Staubli VAL3: loadTemplate.pgx

program loadTemplate()
begin
  // load the default instruction
  events:libLoad("Disk://..//templates/instruction")
  delay(0)
end
